PROGRAM SensorsMain
VAR
	
	angleDir : LREAL;
	

	
	sensor_D AT %Q* : BOOL;
	sensor_E AT %Q* : BOOL;
	sensor_F AT %Q* : BOOL;
	
	
	
	
	en_sensor_D AT %Q* : BOOL ;
	en_sensor_E AT %Q* : BOOL ;
	en_sensor_F AT %Q* : BOOL ;


	sensor1_UO1 AT %I* : BOOL;
	sensor1_UO2 AT %I* : BOOL;
	sensor1_UO3 AT %I* : BOOL;
	
	sensor2_UO1 AT %I* : BOOL;
	sensor2_UO2 AT %I* : BOOL;
	sensor2_UO3 AT %I* : BOOL;
	
	tmr1 : TON; //program period
	new_direction : INT := 0; //new direction based on velocity direction
	direction : ARRAY [0..8] OF INT := [0,0,0,0,0,0,0,0,0]; //stock last new directions
	lastChange : LREAL := 0; //prevent to change fields too quickly 
	Index : INT := 0;
	maxVal : INT := -1;
	
	
	
	
	
END_VAR

VAR CONSTANT
	PI_8 : LREAL := 0.39269908169872414;
	VMAX : LREAL := 1.2;
	VTHMAX : LREAL := 0.5;
	TPROG : LREAL := 0.001;
	TWAIT : LREAL := 0.2;
 	

END_VAR

//Compute acctual direction of the mobile platform
IF(ABS(ControlGVL.forwardReverse)<0.04) THEN
	IF(ControlGVL.leftRight>0.04) THEN
		new_direction := DirPlatform.PLUS_Y;
	ELSIF(ControlGVL.leftRight<-0.04) THEN
		new_direction := DirPlatform.MINUS_Y;
	ELSE
		new_direction := DirPlatform.PLUS_X; //assume default field is Plus X
	END_IF

ELSE
	angleDir := ATAN(-ControlGVL.leftRight/ControlGVL.forwardReverse);
	IF(ControlGVL.forwardReverse<0) THEN
		angleDir := angleDir + 3.141592;
	END_IF

	IF((angleDir>=PI_8)AND(angleDir<3*PI_8)) THEN
		new_direction := DirPlatform.PLUS_X_MINUS_Y;
	ELSIF((angleDir>=3*PI_8)AND(angleDir<5*PI_8)) THEN
		new_direction := DirPlatform.MINUS_Y;
	ELSIF((angleDir>=5*PI_8)AND(angleDir<7*PI_8)) THEN
		new_direction := DirPlatform.MINUS_X_MINUS_Y;
	ELSIF((angleDir>=7*PI_8)AND(angleDir<9*PI_8)) THEN
		new_direction := DirPlatform.MINUS_X;
	ELSIF((angleDir>=9*PI_8)AND(angleDir<11*PI_8)) THEN
		new_direction := DirPlatform.MINUS_X_PLUS_Y;
	ELSIF(((angleDir>=11*PI_8)AND(angleDir<12*PI_8))OR((angleDir>=-4*PI_8)AND(angleDir<-3*PI_8))) THEN
		new_direction := DirPlatform.PLUS_Y;
	ELSIF((angleDir>=-3*PI_8)AND(angleDir<-1*PI_8)) THEN
		new_direction := DirPlatform.PLUS_X_PLUS_Y;
	ELSE
		new_direction := DirPlatform.PLUS_X;
	END_IF
END_IF


//prevent to change too often the set of fields
lastChange := lastChange + TPROG;
//store the new_direction of the cycle
direction[new_direction] := direction[new_direction] +1;
IF((lastChange>TWAIT)) THEN //possibly change only each TWAIT seconds
	
	maxVal := -1;
	FOR Index := 0 TO 8 DO //find the direction most asked
		IF direction[Index] > maxVal THEN
			maxVal := direction[Index];
			new_direction := Index;
		END_IF
		//reset variable for another cycle
  		direction[Index] := 0;
	END_FOR

	SensorsGVL.platformDir := new_direction; //update the fields
	lastChange := 0;
END_IF






//emable writting output
en_sensor_D := TRUE;
en_sensor_E := TRUE;
en_sensor_F := TRUE;



//Update fields on sensors
sensor_D := (SensorsGVL.platformDir / 4)>0;
sensor_E := ((SensorsGVL.platformDir MOD 4)/2)>0;
sensor_F := (SensorsGVL.platformDir MOD 2) >0;




//Adapt maximum speed if obstacles
IF (sensor1_UO1 OR sensor2_UO1) THEN
	ControlGVL.currentVelMax := 0;
	ControlGVL.currentThVelMax :=0;
ELSIF (sensor1_UO2 OR sensor2_UO2) THEN
	ControlGVL.currentVelMax := VMAX/4;
	ControlGVL.currentThVelMax :=VTHMAX;
ELSIF (sensor1_UO3 OR sensor2_UO3) THEN
	ControlGVL.currentVelMax := VMAX/2;
	ControlGVL.currentThVelMax :=VTHMAX;
ELSE
	ControlGVL.currentVelMax := VMAX;
	ControlGVL.currentThVelMax :=VTHMAX;
END_IF

ControlGVL.currentVelMax := VMAX/2;
ControlGVL.currentThVelMax :=VTHMAX;

END_PROGRAM

(* stored: Version 1.1.0.1, ProductVersion 3.1.4024.10
   POU SensorsMain: Id {a5b3c758-f6ce-48b5-b926-741f9ad72276}, SpecialFunc None *)
